TYPE DUT_OutInfoOrigin :
STRUCT
	OriginName		: STRING(50);
	NameX			: STRING(10);
	X				: REAL;
	NameY			: STRING(10);
	Y				: REAL;
	NameZ			: STRING(10);
	Z				: REAL;
	NameB			: STRING(10);
	B				: REAL;
END_STRUCT
END_TYPE

(* stored: Version 1.1.0.1, ProductVersion 3.1.4024.15
   DUT DUT_OutInfoOrigin: Id {b6d36dc4-f9c0-4985-ae7e-c4d9309a5a9d} *)
